Staubli VAL3: TRAJ.pjx

--- TRAJ.pjx ---
Parameters version=s7.6.1 stackSize=5000 millimeterUnit=true
Program file=copy_it.pgx
Program file=link_all.pgx
Program file=link_it.pgx
Data file=TRAJ.dtx
Library alias=saveData path=Disk://saveData/savedata.pjx
Type name=Traies path=Disk://kernel/template/Traies/Traies.pjx
Type name=FrameItem path=Disk://kernel/template/FrameItem/FrameItem.pjx

--- TRAJ.dtx ---
public Traies tTraj{}
  [cuigan1]
    frame fFrame = {fatherId=world[0]}
    num nIndexFrame
    num nIndexTool
    string sID = "cuigan1"
    TrajItem tData[7]
      [0]
        num nType
        pointRx pCircle = {fatherId=tTraj["cuigan1"].fFrame[0]}
        pointRx pPoint = {x=-565.01624, y=1084.746072, z=465.835311, rx=179.23959, ry=0.858813, rz=-1.67867, fatherId=tTraj["cuigan1"].fFrame[0]}
        TrajectoryItem tSuper
          [0]
            string comment
            num distance
            InstrItem iInstr[3]
              [0]
                string sData
                string sType
              [1]
                string sData
                string sType
              [2]
                string sData
                string sType
            num moveType = 1
            num nMoveId
            num nStop
            num nTcpAction
            num nTime
            mdesc nom_speed = {vel=450, tmax=1000}
            bool toStop
      [1]
        num nType
        pointRx pCircle = {fatherId=tTraj["cuigan1"].fFrame[0]}
        pointRx pPoint = {x=-565.016272, y=1104.675398, z=311.255081, rx=179.238004, ry=0.859599, rz=-1.678727, fatherId=tTraj["cuigan1"].fFrame[0]}
        TrajectoryItem tSuper
          [0]
            string comment
            num distance
            InstrItem iInstr[3]
              [0]
                string sData
                string sType
              [1]
                string sData
                string sType
              [2]
                string sData
                string sType
            num moveType = 1
            num nMoveId
            num nStop
            num nTcpAction
            num nTime
            mdesc nom_speed = {vel=450, tmax=1000}
            bool toStop
      [2]
        num nType
        pointRx pCircle = {fatherId=tTraj["cuigan1"].fFrame[0]}
        pointRx pPoint = {x=-538.260119, y=1104.810511, z=225.498274, rx=179.237739, ry=0.859834, rz=-1.678613, fatherId=tTraj["cuigan1"].fFrame[0]}
        TrajectoryItem tSuper
          [0]
            string comment
            num distance
            InstrItem iInstr[3]
              [0]
                string sData
                string sType
              [1]
                string sData
                string sType
              [2]
                string sData
                string sType
            num moveType = 1
            num nMoveId
            num nStop
            num nTcpAction
            num nTime
            mdesc nom_speed = {vel=450, tmax=1000}
            bool toStop
      [3]
        num nType
        pointRx pCircle = {fatherId=tTraj["cuigan1"].fFrame[0]}
        pointRx pPoint = {x=-538.317834, y=1104.616637, z=12.416075, rx=179.237938, ry=0.859601, rz=-1.678818, fatherId=tTraj["cuigan1"].fFrame[0]}
        TrajectoryItem tSuper
          [0]
            string comment
            num distance
            InstrItem iInstr[3]
              [0]
                string sData
                string sType
              [1]
                string sData
                string sType
              [2]
                string sData
                string sType
            num moveType = 1
            num nMoveId
            num nStop
            num nTcpAction
            num nTime
            mdesc nom_speed = {vel=450, tmax=1000}
            bool toStop
      [4]
        num nType
        pointRx pCircle = {fatherId=tTraj["cuigan1"].fFrame[0]}
        pointRx pPoint = {x=-538.260119, y=1104.810511, z=225.498274, rx=179.237739, ry=0.859834, rz=-1.678613, fatherId=tTraj["cuigan1"].fFrame[0]}
        TrajectoryItem tSuper
          [0]
            string comment
            num distance
            InstrItem iInstr[3]
              [0]
                string sData
                string sType
              [1]
                string sData
                string sType
              [2]
                string sData
                string sType
            num moveType = 1
            num nMoveId
            num nStop
            num nTcpAction
            num nTime
            mdesc nom_speed = {vel=450, tmax=1000}
            bool toStop
      [5]
        num nType
        pointRx pCircle = {fatherId=tTraj["cuigan1"].fFrame[0]}
        pointRx pPoint = {x=-538.317834, y=1104.616637, z=12.416075, rx=179.237938, ry=0.859601, rz=-1.678818, fatherId=tTraj["cuigan1"].fFrame[0]}
        TrajectoryItem tSuper
          [0]
            string comment
            num distance
            InstrItem iInstr[3]
              [0]
                string sData
                string sType
              [1]
                string sData
                string sType
              [2]
                string sData
                string sType
            num moveType = 1
            num nMoveId
            num nStop
            num nTcpAction
            num nTime
            mdesc nom_speed = {vel=450, tmax=1000}
            bool toStop
      [6]
        num nType
        pointRx pCircle = {fatherId=tTraj["cuigan1"].fFrame[0]}
        pointRx pPoint = {x=-565.016272, y=1104.675398, z=311.255081, rx=179.238004, ry=0.859599, rz=-1.678727, fatherId=tTraj["cuigan1"].fFrame[0]}
        TrajectoryItem tSuper
          [0]
            string comment
            num distance
            InstrItem iInstr[3]
              [0]
                string sData
                string sType
              [1]
                string sData
                string sType
              [2]
                string sData
                string sType
            num moveType = 1
            num nMoveId
            num nStop
            num nTcpAction
            num nTime
            mdesc nom_speed = {vel=450, tmax=1000}
            bool toStop
  [cuigan2]
    frame fFrame = {fatherId=world[0]}
    num nIndexFrame
    num nIndexTool
    string sID = "cuigan2"
    TrajItem tData[6]
      [0]
        num nType
        pointRx pCircle = {fatherId=tTraj["cuigan2"].fFrame[0]}
        pointRx pPoint = {x=51.287795, y=619.94646, z=-194.31333, rx=-89.153335, ry=-0.841876, rz=179.561969, fatherId=tTraj["cuigan2"].fFrame[0]}
        TrajectoryItem tSuper
          [0]
            string comment
            num distance
            InstrItem iInstr[3]
              [0]
                string sData
                string sType
              [1]
                string sData
                string sType
              [2]
                string sData
                string sType
            num moveType = 1
            num nMoveId
            num nStop
            num nTcpAction
            num nTime
            mdesc nom_speed = {vel=450, tmax=1000}
            bool toStop
      [1]
        num nType
        pointRx pCircle = {fatherId=tTraj["cuigan2"].fFrame[0]}
        pointRx pPoint = {x=90.039083, y=1344.734275, z=-194.313332, rx=-89.152927, ry=-0.841045, rz=179.561766, fatherId=tTraj["cuigan2"].fFrame[0]}
        TrajectoryItem tSuper
          [0]
            string comment
            num distance
            InstrItem iInstr[3]
              [0]
                string sData
                string sType
              [1]
                string sData
                string sType
              [2]
                string sData
                string sType
            num moveType = 1
            num nMoveId
            num nStop
            num nTcpAction
            num nTime
            mdesc nom_speed = {vel=450, tmax=1000}
            bool toStop
      [2]
        num nType
        pointRx pCircle = {fatherId=tTraj["cuigan2"].fFrame[0]}
        pointRx pPoint = {x=106.559445, y=1356.824362, z=-208.795382, rx=-89.14348, ry=-0.832274, rz=-179.80253, fatherId=tTraj["cuigan2"].fFrame[0]}
        TrajectoryItem tSuper
          [0]
            string comment
            num distance
            InstrItem iInstr[3]
              [0]
                string sData
                string sType
              [1]
                string sData
                string sType
              [2]
                string sData
                string sType
            num moveType = 1
            num nMoveId
            num nStop
            num nTcpAction
            num nTime
            mdesc nom_speed = {vel=450, tmax=200, blend=off}
            bool toStop
      [3]
        num nType
        pointRx pCircle = {fatherId=tTraj["cuigan2"].fFrame[0]}
        pointRx pPoint = {x=106.559446, y=1356.82438, z=-337.335235, rx=-89.144125, ry=-0.832423, rz=-179.802189, fatherId=tTraj["cuigan2"].fFrame[0]}
        TrajectoryItem tSuper
          [0]
            string comment
            num distance
            InstrItem iInstr[3]
              [0]
                string sData = "valve1>ON AND valve1>ON"
                string sType = "OUT"
              [1]
                string sData
                string sType
              [2]
                string sData
                string sType
            num moveType = 1
            num nMoveId
            num nStop = 3
            num nTcpAction
            num nTime
            mdesc nom_speed = {vel=450, tmax=200, blend=off}
            bool toStop = true
      [4]
        num nType
        pointRx pCircle = {fatherId=tTraj["cuigan2"].fFrame[0]}
        pointRx pPoint = {x=106.559445, y=1356.824377, z=-314.767495, rx=-89.143975, ry=-0.832401, rz=-179.802206, fatherId=tTraj["cuigan2"].fFrame[0]}
        TrajectoryItem tSuper
          [0]
            string comment
            num distance
            InstrItem iInstr[3]
              [0]
                string sData
                string sType
              [1]
                string sData
                string sType
              [2]
                string sData
                string sType
            num moveType = 1
            num nMoveId
            num nStop
            num nTcpAction
            num nTime
            mdesc nom_speed = {vel=450, tmax=1000, blend=off}
            bool toStop
      [5]
        num nType
        pointRx pCircle = {fatherId=tTraj["cuigan2"].fFrame[0]}
        pointRx pPoint = {x=106.559429, y=861.169145, z=-314.803156, rx=-89.145002, ry=-0.832125, rz=-179.801634, fatherId=tTraj["cuigan2"].fFrame[0]}
        TrajectoryItem tSuper
          [0]
            string comment
            num distance
            InstrItem iInstr[3]
              [0]
                string sData = "valve1>OFF"
                string sType = "OUT"
              [1]
                string sData
                string sType
              [2]
                string sData
                string sType
            num moveType = 1
            num nMoveId
            num nStop = 2
            num nTcpAction
            num nTime
            mdesc nom_speed = {vel=450, tmax=1000, blend=off}
            bool toStop = true
  [langyong]
    frame fFrame = {fatherId=world[0]}
    num nIndexFrame
    num nIndexTool
    string sID = "langyong"
    TrajItem tData[17]
      [0]
        num nType
        pointRx pCircle = {fatherId=tTraj["langyong"].fFrame[0]}
        pointRx pPoint = {x=101.406952, y=-672.049929, z=134.482759, rx=0.234339, ry=-179.225552, rz=-0.433983, fatherId=tTraj["langyong"].fFrame[0]}
        TrajectoryItem tSuper
          [0]
            string comment
            num distance
            InstrItem iInstr[3]
              [0]
                string sData
                string sType
              [1]
                string sData
                string sType
              [2]
                string sData
                string sType
            num moveType = 1
            num nMoveId
            num nStop
            num nTcpAction
            num nTime
            mdesc nom_speed = {vel=450, tmax=1000}
            bool toStop
      [1]
        num nType
        pointRx pCircle = {fatherId=tTraj["langyong"].fFrame[0]}
        pointRx pPoint = {x=101.406944, y=-672.049878, z=728.441619, rx=0.23343, ry=-179.225713, rz=-0.433988, fatherId=tTraj["langyong"].fFrame[0]}
        TrajectoryItem tSuper
          [0]
            string comment
            num distance
            InstrItem iInstr[3]
              [0]
                string sData
                string sType
              [1]
                string sData
                string sType
              [2]
                string sData
                string sType
            num moveType = 1
            num nMoveId
            num nStop
            num nTcpAction
            num nTime
            mdesc nom_speed = {vel=450, tmax=1000}
            bool toStop
      [2]
        num nType
        pointRx pCircle = {fatherId=tTraj["langyong"].fFrame[0]}
        pointRx pPoint = {x=-1006.192711, y=-321.924635, z=728.386217, rx=0.773632, ry=179.762032, rz=89.809237, fatherId=tTraj["langyong"].fFrame[0]}
        TrajectoryItem tSuper
          [0]
            string comment
            num distance
            InstrItem iInstr[3]
              [0]
                string sData
                string sType
              [1]
                string sData
                string sType
              [2]
                string sData
                string sType
            num moveType = 1
            num nMoveId
            num nStop
            num nTcpAction
            num nTime
            mdesc nom_speed = {vel=450, tmax=1000}
            bool toStop
      [3]
        num nType
        pointRx pCircle = {fatherId=tTraj["langyong"].fFrame[0]}
        pointRx pPoint = {x=-1006.192699, y=-321.924631, z=182.66322, rx=0.773882, ry=179.761186, rz=89.809222, fatherId=tTraj["langyong"].fFrame[0]}
        TrajectoryItem tSuper
          [0]
            string comment
            num distance
            InstrItem iInstr[3]
              [0]
                string sData
                string sType
              [1]
                string sData
                string sType
              [2]
                string sData
                string sType
            num moveType = 1
            num nMoveId
            num nStop
            num nTcpAction
            num nTime
            mdesc nom_speed = {vel=450, tmax=1000}
            bool toStop
      [4]
        num nType
        pointRx pCircle = {fatherId=tTraj["langyong"].fFrame[0]}
        pointRx pPoint = {x=-1281.375139, y=-321.924578, z=182.721178, rx=0.773404, ry=179.763035, rz=89.809305, fatherId=tTraj["langyong"].fFrame[0]}
        TrajectoryItem tSuper
          [0]
            string comment
            num distance
            InstrItem iInstr[3]
              [0]
                string sData
                string sType
              [1]
                string sData
                string sType
              [2]
                string sData
                string sType
            num moveType = 1
            num nMoveId
            num nStop
            num nTcpAction
            num nTime
            mdesc nom_speed = {vel=450, tmax=1000}
            bool toStop
      [5]
        num nType
        pointRx pCircle = {fatherId=tTraj["langyong"].fFrame[0]}
        pointRx pPoint = {x=-1145.724954, y=-423.872189, z=182.721219, rx=0.773033, ry=179.761848, rz=89.808331, fatherId=tTraj["langyong"].fFrame[0]}
        TrajectoryItem tSuper
          [0]
            string comment
            num distance
            InstrItem iInstr[3]
              [0]
                string sData
                string sType
              [1]
                string sData
                string sType
              [2]
                string sData
                string sType
            num moveType = 1
            num nMoveId
            num nStop
            num nTcpAction
            num nTime
            mdesc nom_speed = {vel=450, tmax=1000}
            bool toStop
      [6]
        num nType
        pointRx pCircle = {fatherId=tTraj["langyong"].fFrame[0]}
        pointRx pPoint = {x=-1145.724991, y=-190.623351, z=182.721231, rx=0.774211, ry=179.761503, rz=89.809834, fatherId=tTraj["langyong"].fFrame[0]}
        TrajectoryItem tSuper
          [0]
            string comment
            num distance
            InstrItem iInstr[3]
              [0]
                string sData
                string sType
              [1]
                string sData
                string sType
              [2]
                string sData
                string sType
            num moveType = 1
            num nMoveId
            num nStop
            num nTcpAction
            num nTime
            mdesc nom_speed = {vel=450, tmax=1000}
            bool toStop
      [7]
        num nType
        pointRx pCircle = {fatherId=tTraj["langyong"].fFrame[0]}
        pointRx pPoint = {x=-1145.724949, y=-291.394683, z=182.721226, rx=0.773733, ry=179.761744, rz=89.809222, fatherId=tTraj["langyong"].fFrame[0]}
        TrajectoryItem tSuper
          [0]
            string comment
            num distance
            InstrItem iInstr[3]
              [0]
                string sData
                string sType
              [1]
                string sData
                string sType
              [2]
                string sData
                string sType
            num moveType = 1
            num nMoveId
            num nStop
            num nTcpAction
            num nTime
            mdesc nom_speed = {vel=450, tmax=1000, blend=off}
            bool toStop
      [8]
        num nType
        pointRx pCircle = {fatherId=tTraj["langyong"].fFrame[0]}
        pointRx pPoint = {x=-1145.724431, y=-291.336847, z=774.025897, rx=0.773928, ry=179.762576, rz=89.809844, fatherId=tTraj["langyong"].fFrame[0]}
        TrajectoryItem tSuper
          [0]
            string comment
            num distance
            InstrItem iInstr[3]
              [0]
                string sData
                string sType
              [1]
                string sData
                string sType
              [2]
                string sData
                string sType
            num moveType = 1
            num nMoveId
            num nStop
            num nTcpAction
            num nTime
            mdesc nom_speed = {vel=450, tmax=1000, blend=off}
            bool toStop
      [9]
        num nType
        pointRx pCircle = {fatherId=tTraj["langyong"].fFrame[0]}
        pointRx pPoint = {x=-616.214813, y=-291.336879, z=774.025978, rx=113.876013, ry=-87.910341, rz=-68.457504, fatherId=tTraj["langyong"].fFrame[0]}
        TrajectoryItem tSuper
          [0]
            string comment
            num distance
            InstrItem iInstr[3]
              [0]
                string sData
                string sType
              [1]
                string sData
                string sType
              [2]
                string sData
                string sType
            num moveType = 1
            num nMoveId
            num nStop
            num nTcpAction
            num nTime
            mdesc nom_speed = {vel=450, tmax=1000, blend=off}
            bool toStop
      [10]
        num nType
        pointRx pCircle = {fatherId=tTraj["langyong"].fFrame[0]}
        pointRx pPoint = {x=-616.216294, y=-291.337814, z=451.093035, rx=113.907266, ry=-87.909592, rz=-68.426624, fatherId=tTraj["langyong"].fFrame[0]}
        TrajectoryItem tSuper
          [0]
            string comment
            num distance
            InstrItem iInstr[3]
              [0]
                string sData
                string sType
              [1]
                string sData
                string sType
              [2]
                string sData
                string sType
            num moveType = 1
            num nMoveId
            num nStop
            num nTcpAction
            num nTime
            mdesc nom_speed = {vel=450, tmax=1000, blend=off}
            bool toStop
      [11]
        num nType
        pointRx pCircle = {fatherId=tTraj["langyong"].fFrame[0]}
        pointRx pPoint = {x=-616.216319, y=-930.694647, z=451.150628, rx=-144.54891, ry=-89.320818, rz=34.963724, fatherId=tTraj["langyong"].fFrame[0]}
        TrajectoryItem tSuper
          [0]
            string comment
            num distance
            InstrItem iInstr[3]
              [0]
                string sData
                string sType
              [1]
                string sData
                string sType
              [2]
                string sData
                string sType
            num moveType = 1
            num nMoveId
            num nStop
            num nTcpAction
            num nTime
            mdesc nom_speed = {vel=450, tmax=1000, blend=off}
            bool toStop
      [12]
        num nType
        pointRx pCircle = {fatherId=tTraj["langyong"].fFrame[0]}
        pointRx pPoint = {x=-733.462537, y=-948.698758, z=451.150628, rx=-144.392076, ry=-89.320484, rz=35.120439, fatherId=tTraj["langyong"].fFrame[0]}
        TrajectoryItem tSuper
          [0]
            string comment
            num distance
            InstrItem iInstr[3]
              [0]
                string sData
                string sType
              [1]
                string sData
                string sType
              [2]
                string sData
                string sType
            num moveType = 1
            num nMoveId
            num nStop
            num nTcpAction
            num nTime
            mdesc nom_speed = {vel=450, tmax=1000, blend=off}
            bool toStop
      [13]
        num nType
        pointRx pCircle = {fatherId=tTraj["langyong"].fFrame[0]}
        pointRx pPoint = {x=-733.46251, y=-948.753526, z=789.250968, rx=-144.409498, ry=-89.320655, rz=35.103658, fatherId=tTraj["langyong"].fFrame[0]}
        TrajectoryItem tSuper
          [0]
            string comment
            num distance
            InstrItem iInstr[3]
              [0]
                string sData
                string sType
              [1]
                string sData
                string sType
              [2]
                string sData
                string sType
            num moveType = 1
            num nMoveId
            num nStop
            num nTcpAction
            num nTime
            mdesc nom_speed = {vel=450, tmax=1000, blend=off}
            bool toStop
      [14]
        num nType
        pointRx pCircle = {fatherId=tTraj["langyong"].fFrame[0]}
        pointRx pPoint = {x=-733.462551, y=-948.753601, z=458.650073, rx=-144.453108, ry=-89.319, rz=35.059012, fatherId=tTraj["langyong"].fFrame[0]}
        TrajectoryItem tSuper
          [0]
            string comment
            num distance
            InstrItem iInstr[3]
              [0]
                string sData
                string sType
              [1]
                string sData
                string sType
              [2]
                string sData
                string sType
            num moveType = 1
            num nMoveId
            num nStop
            num nTcpAction
            num nTime
            mdesc nom_speed = {vel=450, tmax=1000, blend=off}
            bool toStop
      [15]
        num nType
        pointRx pCircle = {fatherId=tTraj["langyong"].fFrame[0]}
        pointRx pPoint = {x=-161.262092, y=-948.753567, z=458.708003, rx=-144.464792, ry=-89.320196, rz=35.047398, fatherId=tTraj["langyong"].fFrame[0]}
        TrajectoryItem tSuper
          [0]
            string comment
            num distance
            InstrItem iInstr[3]
              [0]
                string sData
                string sType
              [1]
                string sData
                string sType
              [2]
                string sData
                string sType
            num moveType = 1
            num nMoveId
            num nStop
            num nTcpAction
            num nTime
            mdesc nom_speed = {vel=450, tmax=1000, blend=off}
            bool toStop
      [16]
        num nType
        pointRx pCircle = {fatherId=tTraj["langyong"].fFrame[0]}
        pointRx pPoint = {x=-161.31928, y=-948.753617, z=458.708043, rx=-179.603947, ry=-1.154201, rz=-0.477431, fatherId=tTraj["langyong"].fFrame[0]}
        TrajectoryItem tSuper
          [0]
            string comment
            num distance
            InstrItem iInstr[3]
              [0]
                string sData
                string sType
              [1]
                string sData
                string sType
              [2]
                string sData
                string sType
            num moveType = 1
            num nMoveId
            num nStop
            num nTcpAction
            num nTime
            mdesc nom_speed = {vel=450, tmax=1000, blend=off}
            bool toStop
  [qujian]
    frame fFrame = {fatherId=world[0]}
    num nIndexFrame
    num nIndexTool
    string sID = "qujian"
    TrajItem tData[6]
      [0]
        num nType
        pointRx pCircle = {fatherId=tTraj["qujian"].fFrame[0]}
        pointRx pPoint = {x=105.007696, y=-816.81224, z=-359.969919, rx=-89.572329, ry=-179.228248, rz=-0.110408, fatherId=tTraj["qujian"].fFrame[0]}
        TrajectoryItem tSuper
          [0]
            string comment
            num distance
            InstrItem iInstr[3]
              [0]
                string sData = "valve1>ON"
                string sType = "OUT"
              [1]
                string sData
                string sType
              [2]
                string sData
                string sType
            num moveType = 1
            num nMoveId
            num nStop = 2
            num nTcpAction
            num nTime
            mdesc nom_speed = {vel=450, tmax=1000, blend=off}
            bool toStop = true
      [1]
        num nType
        pointRx pCircle = {fatherId=tTraj["qujian"].fFrame[0]}
        pointRx pPoint = {x=104.982849, y=-1429.69004, z=-358.03106, rx=-89.573114, ry=-179.2277, rz=-0.109849, fatherId=tTraj["qujian"].fFrame[0]}
        TrajectoryItem tSuper
          [0]
            string comment
            num distance
            InstrItem iInstr[3]
              [0]
                string sData
                string sType
              [1]
                string sData
                string sType
              [2]
                string sData
                string sType
            num moveType = 1
            num nMoveId
            num nStop
            num nTcpAction
            num nTime
            mdesc nom_speed = {vel=450, tmax=1000, blend=off}
            bool toStop
      [2]
        num nType
        pointRx pCircle = {fatherId=tTraj["qujian"].fFrame[0]}
        pointRx pPoint = {x=101.407856, y=-1425.629051, z=-323.450838, rx=-89.577502, ry=-179.225148, rz=-0.433251, fatherId=tTraj["qujian"].fFrame[0]}
        TrajectoryItem tSuper
          [0]
            string comment
            num distance
            InstrItem iInstr[3]
              [0]
                string sData = "valve1>OFF"
                string sType = "OUT"
              [1]
                string sData
                string sType
              [2]
                string sData
                string sType
            num moveType = 1
            num nMoveId
            num nStop = 3
            num nTcpAction = -2
            num nTime
            mdesc nom_speed = {vel=450, tmax=200, blend=off}
            bool toStop = true
      [3]
        num nType
        pointRx pCircle = {fatherId=tTraj["qujian"].fFrame[0]}
        pointRx pPoint = {x=101.407529, y=-1425.628022, z=-202.340179, rx=-89.578087, ry=-179.225456, rz=-0.433081, fatherId=tTraj["qujian"].fFrame[0]}
        TrajectoryItem tSuper
          [0]
            string comment
            num distance
            InstrItem iInstr[3]
              [0]
                string sData
                string sType
              [1]
                string sData
                string sType
              [2]
                string sData
                string sType
            num moveType = 1
            num nMoveId
            num nStop = 3
            num nTcpAction = -2
            num nTime
            mdesc nom_speed = {vel=450, tmax=200, blend=off}
            bool toStop
      [4]
        num nType
        pointRx pCircle = {fatherId=tTraj["qujian"].fFrame[0]}
        pointRx pPoint = {x=101.407495, y=-672.050967, z=-202.398205, rx=-89.576621, ry=-179.2256, rz=-0.433991, fatherId=tTraj["qujian"].fFrame[0]}
        TrajectoryItem tSuper
          [0]
            string comment
            num distance
            InstrItem iInstr[3]
              [0]
                string sData
                string sType
              [1]
                string sData
                string sType
              [2]
                string sData
                string sType
            num moveType = 1
            num nMoveId
            num nStop
            num nTcpAction = -2
            num nTime
            mdesc nom_speed = {vel=450, tmax=1000, blend=off}
            bool toStop
      [5]
        num nType
        pointRx pCircle = {fatherId=tTraj["qujian"].fFrame[0]}
        pointRx pPoint = {x=101.40751, y=-672.050938, z=134.485123, rx=0.233988, ry=-179.22561, rz=-0.433995, fatherId=tTraj["qujian"].fFrame[0]}
        TrajectoryItem tSuper
          [0]
            string comment
            num distance
            InstrItem iInstr[3]
              [0]
                string sData
                string sType
              [1]
                string sData
                string sType
              [2]
                string sData
                string sType
            num moveType = 1
            num nMoveId
            num nStop
            num nTcpAction = -2
            num nTime
            mdesc nom_speed = {vel=450, tmax=1000, blend=off}
            bool toStop
  [test]
    frame fFrame = {fatherId=world[0]}
    num nIndexFrame
    num nIndexTool
    string sID = "test"
    TrajItem tData[7]
      [0]
        num nType
        pointRx pCircle = {fatherId=tTraj["test"].fFrame[0]}
        pointRx pPoint = {x=1198, y=151.559856, z=210.59, rx=87.981257, ry=172.229649, rz=-80.060298, fatherId=tTraj["test"].fFrame[0]}
        TrajectoryItem tSuper
          [0]
            string comment
            num distance
            InstrItem iInstr[3]
              [0]
                string sData
                string sType
              [1]
                string sData
                string sType
              [2]
                string sData
                string sType
            num moveType = 1
            num nMoveId
            num nStop
            num nTcpAction
            num nTime
            mdesc nom_speed = {accel=200, vel=450, decel=200, tmax=2000}
            bool toStop
      [1]
        num nType
        pointRx pCircle = {fatherId=tTraj["test"].fFrame[0]}
        pointRx pPoint = {x=2198.708273, y=151.559856, z=210.59, rx=87.981257, ry=172.229649, rz=-80.060298, fatherId=tTraj["test"].fFrame[0]}
        TrajectoryItem tSuper
          [0]
            string comment
            num distance
            InstrItem iInstr[3]
              [0]
                string sData
                string sType
              [1]
                string sData
                string sType
              [2]
                string sData
                string sType
            num moveType = 1
            num nMoveId
            num nStop
            num nTcpAction
            num nTime
            mdesc nom_speed = {accel=200, vel=450, decel=200, tmax=2000, leave=30, reach=30}
            bool toStop
      [2]
        num nType
        pointRx pCircle = {fatherId=tTraj["test"].fFrame[0]}
        pointRx pPoint = {x=2198.708273, y=151.559856, z=410.59, rx=87.981257, ry=172.229649, rz=-80.060298, fatherId=tTraj["test"].fFrame[0]}
        TrajectoryItem tSuper
          [0]
            string comment = "shangtai"
            num distance
            InstrItem iInstr[3]
              [0]
                string sData
                string sType
              [1]
                string sData
                string sType
              [2]
                string sData
                string sType
            num moveType = 1
            num nMoveId
            num nStop
            num nTcpAction
            num nTime
            mdesc nom_speed = {accel=200, vel=450, decel=200, tmax=2000, leave=30, reach=30}
            bool toStop
      [3]
        num nType
        pointRx pCircle = {fatherId=tTraj["test"].fFrame[0]}
        pointRx pPoint = {x=2298.71, y=251.56, z=410.59, rx=87.981257, ry=172.229649, rz=-80.060298, fatherId=tTraj["test"].fFrame[0]}
        TrajectoryItem tSuper
          [0]
            string comment = "daoda"
            num distance
            InstrItem iInstr[3]
              [0]
                string sData
                string sType
              [1]
                string sData
                string sType
              [2]
                string sData
                string sType
            num moveType = 1
            num nMoveId
            num nStop = 1.5
            num nTcpAction
            num nTime
            mdesc nom_speed = {vel=450, tmax=500, blend=off}
            bool toStop = true
      [4]
        num nType
        pointRx pCircle = {fatherId=tTraj["test"].fFrame[0]}
        pointRx pPoint = {x=2198.708273, y=151.559856, z=410.59, rx=87.981257, ry=172.229649, rz=-80.060298, fatherId=tTraj["test"].fFrame[0]}
        TrajectoryItem tSuper
          [0]
            string comment = "xiajiang"
            num distance
            InstrItem iInstr[3]
              [0]
                string sData
                string sType
              [1]
                string sData
                string sType
              [2]
                string sData
                string sType
            num moveType = 1
            num nMoveId
            num nStop = 1.5
            num nTcpAction
            num nTime
            mdesc nom_speed = {accel=200, vel=450, decel=200, tmax=2000, blend=off}
            bool toStop
      [5]
        num nType
        pointRx pCircle = {fatherId=tTraj["test"].fFrame[0]}
        pointRx pPoint = {x=2198.708273, y=151.559856, z=210.59, rx=87.981257, ry=172.229649, rz=-80.060298, fatherId=tTraj["test"].fFrame[0]}
        TrajectoryItem tSuper
          [0]
            string comment
            num distance
            InstrItem iInstr[3]
              [0]
                string sData
                string sType
              [1]
                string sData
                string sType
              [2]
                string sData
                string sType
            num moveType = 1
            num nMoveId
            num nStop
            num nTcpAction
            num nTime
